(* IEC 61131-3 sources: eCockpitGit/test_project/src/%F%00 Library/%F%Common Functions/%F%String/%F%Normal/%F%Find, 3 files *)

(* ---- %POU%FU_wFind.st ---- *)
//This function, returns the lenght of a string
// |**Version**|**Author**| **Date** |**Changes**
// | 1         | NSN      | 13-06-18 | Creation
FUNCTION FU_wFind : WORD
VAR_INPUT
	s1			:STRING(255);		//Input String1
	s2			:STRING(255);		//Input String2
END_VAR
(*%!%__DELIMITER__%!%*)
FU_wFind	:=		FU_wFindBI(s1:=s1,s2:=s2);

(* ---- %POU%FU_wFindRight.st ---- *)
//This function, returns the lenght of a string
// |**Version**|**Author**| **Date** |**Changes**
// | 1         | NSN      | 13-06-18 | Creation
FUNCTION FU_wFindRight : WORD
VAR_INPUT
	s1			:STRING(255);		//Input String1
	s2			:STRING(255);		//Input String2
END_VAR
(*%!%__DELIMITER__%!%*)
FU_wFindRight	:=		FU_wFindRightBI(s1:=s1,s2:=s2);

(* ---- %POU%FU_wFindSkip.st ---- *)
//This function, returns the lenght of a string
// |**Version**|**Author**| **Date** |**Changes**
// | 1         | NSN      | 13-06-18 | Creation
FUNCTION FU_wFindSkip : WORD
VAR_INPUT
	s1			:STRING(255);		//Input String1
	s2			:STRING(255);		//Input String2
	skipAmount	:BYTE;				//Amount to skip
END_VAR
(*%!%__DELIMITER__%!%*)
FU_wFindSkip	:=		FU_wFindSkipBI(s1:=s1,s2:=s2,skipAmount:=skipAmount);
